// TIA Portal V16 export
// export: Created 2024-12-03T15:41:42.4438673Z, ExportSetting WithDefaults, DisplayName Totally Integrated Automation Portal, DisplayVersion V16 Update 6, DisplayName TIA Portal Version Control Interface, DisplayVersion V16 Update 2, DisplayName TIA Portal Openness, DisplayVersion V16 Update 6, DisplayName TIA Portal Teamcenter Gateway, DisplayVersion V16, DisplayName SINAMICS Startdrive Advanced, DisplayVersion V16 Update 5, DisplayName SINAMICS Startdrive G130, G150, S120, S150, SINAMICS MV, S210, DisplayVersion V16 Update 5, DisplayName SINAMICS Startdrive G110M, G120, G120C, G120D, G120P, G115D, DisplayVersion V16 Update 5, DisplayName STEP 7 Professional, DisplayVersion V16 Update 6, DisplayName STEP 7 Safety, DisplayVersion V16, DisplayName WinCC Advanced / Unified PC, DisplayVersion V16 Update 6
FUNCTION_BLOCK "EC_Cognex_Dataman_Single_FB"   // FB84, SCL
{ S7_Optimized_Access := 'TRUE' }
VERSION : 0.1
// stored: AutoNumber true, IsIECCheckEnabled false, IsRetainMemResEnabled false, MemoryReserve 100, SetENOAutomatically false, UDAEnableTagReadback false
   VAR_INPUT
      I_HwId : HW_ANY;
      I_Result : "COGNEX_DATAMAN_IN_RESULT_UDT";
      I_ResultStatus : "COGNEX_DATAMAN_IN_RESULT_STATUS_UDT";
      I_Status : "COGNEX_DATAMAN_IN_STATUS_UDT";
   END_VAR
   VAR_OUTPUT
      O_Control : "COGNEX_DATAMAN_OUT_CONTROL_UDT";
      O_Trigger : "COGNEX_DATAMAN_OUT_TRIGGER_UDT";
   END_VAR
   VAR_IN_OUT
      IO_Scanner : "COGNEX_DATAMAN_LOGIC_UDT";
   END_VAR
   VAR
      PrevScanId : Int;
      ScanCommand : "SmartBool";
      triggerAuto { S7_SetPoint := 'True'} : "SmartBool";
      triggerManual { S7_SetPoint := 'True'} : "SmartBool";
      NewResultFlag { S7_SetPoint := 'True'} : "SmartBool";
      MissedTrigger { S7_SetPoint := 'True'} : "SmartBool";
      NotConnected { S7_SetPoint := 'True'} : TON_TIME;
      TimeOutDetector { S7_SetPoint := 'True'} : TON_TIME;
      TimeOutTime { S7_SetPoint := 'True'} : Time;
      StartTimeOut { S7_SetPoint := 'True'} : Bool;
      LockReceiveResult : Bool;
      cycleRun { S7_SetPoint := 'True'} : "CycleRun";
      alarmInfo : "AlarmInfo_UDT";
      TimeOutAlarm { S7_SetPoint := 'True'} : Program_Alarm;
      TriggerGuardAlarm { S7_SetPoint := 'True'} : Program_Alarm;
      ScannerNotConnected { S7_SetPoint := 'True'} : Program_Alarm;
      ErrorFromScanner { S7_SetPoint := 'True'} : Program_Alarm;
      SerialBufferOverlfow { S7_SetPoint := 'True'} : Program_Alarm;
   END_VAR
   VAR_TEMP
      T_AppState : "ApplicationState_UDT";
      T_Zone : "ZoneInfo";
      T_NewResult : Bool;
      T_Error : Int;
      dummy : Array[0..5] of Byte;
   END_VAR
BEGIN
   REGION APPSTATE
       #T_Zone := "ApplicationState_DB".ZoneNames[#IO_Scanner.Zone];
       #T_AppState := "ApplicationState_DB".Appstate[#T_Zone.AppStateIndex];
       #cycleRun();
   END_REGION

   REGION STATUS READERS
       #MissedTrigger(I_Sensor := #I_Status.MissedAck);
       #NewResultFlag(I_Sensor := #I_ResultStatus.ResultsAvaileble);
   END_REGION

   REGION Commands

       #triggerAuto(I_Sensor := #IO_Scanner.Cmd.ScanAuto AND #T_AppState.States.AutoModeActivated.State);
       #triggerManual(I_Sensor := #IO_Scanner.Cmd.ScanManual AND #T_AppState.States.ManualModeActivated.State);

       #ScanCommand(I_Sensor := #triggerAuto.O_data.State OR #triggerManual.O_data.State AND NOT #StartTimeOut);

       IF #ScanCommand.O_data.LE AND NOT #StartTimeOut THEN
           #PrevScanId.%B0 := #I_Status.TriggerId_MSB;
           #PrevScanId.%B1 := #I_Status.TriggerId_LSB;
           #PrevScanId := #PrevScanId;
       END_IF;

   END_REGION

   REGION ALARMS

       REGION INIT
           IF NOT #alarmInfo.init OR #IO_Scanner.Name = '' OR #alarmInfo.info = '' OR "HMI_DB".ReloadSettings.signal THEN
               #alarmInfo.init := true;
               #IO_Scanner.Name := "buildObjectName"(I_Symbolname := GetSymbolName(variable := #IO_Scanner, size := 40));
               #alarmInfo.info := "buildAlarmInfo"(I_ZoneIndex := #IO_Scanner.Zone, I_ZoneName := #T_Zone.ZoneName, I_ObjectName := #IO_Scanner.Name);
           END_IF;
       END_REGION

       REGION timeout scanning
           IF #IO_Scanner.ReadingResult.TimeOut_Pulse THEN
               #IO_Scanner.Alarms.TimeOutReading.Active := TRUE;
           END_IF;
           #IO_Scanner.Alarms.TimeOutReading.Active := FALSE;
           #IO_Scanner.Alarms.status.%X0 := #IO_Scanner.Alarms.TimeOutReading.Active;
       END_REGION

       REGION trigger guard
           IF (#triggerAuto.O_data.State
               OR #triggerManual.O_data.State)
               AND #StartTimeOut THEN
               #IO_Scanner.Alarms.TriggerGuard.Active := TRUE;
           END_IF;
           #IO_Scanner.Alarms.status.%X1 := #IO_Scanner.Alarms.TriggerGuard.Active;
       END_REGION

       REGION scanner not connected

           #T_Error := DPRD_DAT(LADDR := #I_HwId, RECORD => #dummy);

           IF #T_Error > 0 THEN
               #IO_Scanner.Alarms.NotConnected.Active := TRUE;
           END_IF;

           #IO_Scanner.Alarms.status.%X2 := #IO_Scanner.Alarms.NotConnected.Active;
       END_REGION

       REGION error from scanner
           IF #I_ResultStatus.GeneralError THEN
               #IO_Scanner.Alarms.ErrorFromScanner.Active := TRUE;
           END_IF;
           #IO_Scanner.Alarms.ErrorFromScanner.Active := FALSE;
           #IO_Scanner.Alarms.status.%X3 := #IO_Scanner.Alarms.ErrorFromScanner.Active;
       END_REGION

       REGION SERIAL BUFFER OVERFLOW
           IF #I_ResultStatus.ResultBufferOverrun THEN
               #IO_Scanner.Alarms.SerialBufferOverFlow.Active := TRUE;
           END_IF;
           #IO_Scanner.Alarms.status.%X4 := #IO_Scanner.Alarms.SerialBufferOverFlow.Active;
       END_REGION

       REGION PROGRAM ALARMS
           IF #cycleRun.O_Cycle = 5 THEN
               #TimeOutAlarm(SIG := #IO_Scanner.Alarms.TimeOutReading.Active,
                             SD_1 := #T_Zone.ZoneName,
                             SD_2 := #IO_Scanner.Name,
                             SD_3 := #alarmInfo.info);
           END_IF;

           IF #cycleRun.O_Cycle = 6 THEN
               #TriggerGuardAlarm(SIG := #IO_Scanner.Alarms.TriggerGuard.Active,
                                  SD_1 := #T_Zone.ZoneName,
                                  SD_2 := #IO_Scanner.Name,
                                  SD_3 := #alarmInfo.info);
           END_IF;

           IF #cycleRun.O_Cycle = 7 THEN
               #ScannerNotConnected(SIG := #IO_Scanner.Alarms.NotConnected.Active,
                                    SD_1 := #T_Zone.ZoneName,
                                    SD_2 := #IO_Scanner.Name,
                                    SD_3 := #alarmInfo.info);
           END_IF;

           IF #cycleRun.O_Cycle = 8 THEN
               #ErrorFromScanner(SIG := #IO_Scanner.Alarms.ErrorFromScanner.Active,
                                 SD_1 := #T_Zone.ZoneName,
                                 SD_2 := #IO_Scanner.Name,
                                 SD_3 := #alarmInfo.info);
           END_IF;

           IF #cycleRun.O_Cycle = 9 THEN
               #SerialBufferOverlfow(SIG := #IO_Scanner.Alarms.SerialBufferOverFlow.Active,
                                     SD_1 := #T_Zone.ZoneName,
                                     SD_2 := #IO_Scanner.Name,
                                     SD_3 := #alarmInfo.info);
           END_IF;

       END_REGION

       IF #IO_Scanner.Alarms.status > 0 THEN
           "ApplicationState_DB".Appstate[#T_Zone.AppStateIndex].Alarms.AlarmActiveInternalPLC := TRUE;
       END_IF;

       IF #T_AppState.Hmi_Buttons.reset.state.State
           OR #IO_Scanner.Cmd.Reset THEN
           #IO_Scanner.Alarms.TimeOutReading.Active := 0;
           #IO_Scanner.Alarms.TriggerGuard.Active := 0;
           #IO_Scanner.Alarms.NotConnected.Active := 0;
           #IO_Scanner.Alarms.ErrorFromScanner.Active := 0;
           #IO_Scanner.Alarms.SerialBufferOverFlow.Active := 0;
       END_IF;

   END_REGION

   REGION Create status

       #IO_Scanner.Status.ManualModeActive := #T_AppState.States.ManualModeActivated.State;
       #IO_Scanner.Status.ReqBusy := #I_ResultStatus.Decoding OR #StartTimeOut;
       #IO_Scanner.Status.ReqDone := NOT #IO_Scanner.Status.ReqBusy;
       #IO_Scanner.Status.ReadyForNewScan := #I_Status.TriggerReady
       AND NOT #ScanCommand.O_data.State;

   END_REGION

   REGION Parse code

       //Reset pulses
       #IO_Scanner.ReadingResult.Barcode_Pulse := '';
       #IO_Scanner.ReadingResult.GoodRead_Pulse := FALSE;
       #IO_Scanner.ReadingResult.BadRead_Pulse := FALSE;
       #IO_Scanner.ReadingResult.TimeOut_Pulse := FALSE;
       #IO_Scanner.ReadingResult.MissedTrigger_Pulse := FALSE;
       #IO_Scanner.ReadingResult.OutOfSync_Pulse := FALSE;
       #IO_Scanner.ReadingResult.NewResult_Pulse := FALSE;

       REGION GOOD READ / BAD READ
           IF #NewResultFlag.O_data.LE
               AND #I_Result.TriggerId = #PrevScanId
               AND NOT #LockReceiveResult THEN

               REGION reset timed out
                   #StartTimeOut := FALSE;
                   #IO_Scanner.ReadingResult.TimeOut := FALSE;
               END_REGION

               REGION Barcode parsing
                   //IF NOT "Simulation_DB".Simulation_On THEN
                   #IO_Scanner.ReadingResult.chars := #I_Result.Barcode;
                   Chars_TO_Strg(Chars := #IO_Scanner.ReadingResult.chars,
                                 pChars := 0,
                                 Cnt := INT_TO_UINT(#I_Result.ResultLength) - 1, //The last char is new line return we don't need this :)
                                 Strg => #IO_Scanner.ReadingResult.Barcode_Pulse);
                   // ELSE
                   //     #IO_Scanner.ReadingResult.Barcode_Pulse := #IO_Scanner.ReadingResult.Barcode;
                   // END_IF;

                   #IO_Scanner.ReadingResult.Barcode := '';
                   #IO_Scanner.ReadingResult.Barcode := #IO_Scanner.ReadingResult.Barcode_Pulse;
               END_REGION

               REGION SIM
                   IF "Simulation_DB".barcode_sim THEN
                       #IO_Scanner.ReadingResult.Barcode_Pulse := 'BarcodeSim';
                       #IO_Scanner.ReadingResult.Barcode := #IO_Scanner.ReadingResult.Barcode_Pulse;
                   END_IF;

               END_REGION

               REGION Good Read / bad read
                   IF #IO_Scanner.ReadingResult.Barcode_Pulse = 'NoRead' THEN
                       #IO_Scanner.ReadingResult.BadRead_Pulse := TRUE;
                   ELSE
                       #IO_Scanner.ReadingResult.GoodRead_Pulse := TRUE;
                   END_IF;
                   #IO_Scanner.ReadingResult.GoodRead := #IO_Scanner.ReadingResult.GoodRead_Pulse;
                   #IO_Scanner.ReadingResult.BadRead := #IO_Scanner.ReadingResult.BadRead_Pulse;
                   #IO_Scanner.ReadingResult.MissedTrigger := FALSE;
                   #IO_Scanner.ReadingResult.OutOfSync := FALSE;
               END_REGION

           END_IF;
       END_REGION

       REGION MISSED TRIGGER
           IF #MissedTrigger.O_data.LE AND NOT #LockReceiveResult THEN
               #IO_Scanner.ReadingResult.GoodRead := FALSE;
               #IO_Scanner.ReadingResult.BadRead := TRUE;
               #IO_Scanner.ReadingResult.MissedTrigger := TRUE;
               #IO_Scanner.ReadingResult.OutOfSync := FALSE;
               #IO_Scanner.ReadingResult.TimeOut := FALSE;

               #IO_Scanner.ReadingResult.MissedTrigger_Pulse := TRUE;

               #IO_Scanner.ReadingResult.Barcode_Pulse := 'MISSED TRIGGER';
               #IO_Scanner.ReadingResult.Barcode := #IO_Scanner.ReadingResult.Barcode_Pulse;
           END_IF;
       END_REGION

       REGION OUT OF SYNC
           IF #NewResultFlag.O_data.LE
               AND #PrevScanId <> #I_Result.TriggerId
               AND NOT #LockReceiveResult
           THEN
               #IO_Scanner.ReadingResult.GoodRead := FALSE;
               #IO_Scanner.ReadingResult.BadRead := TRUE;
               #IO_Scanner.ReadingResult.MissedTrigger := FALSE;
               #IO_Scanner.ReadingResult.OutOfSync := TRUE;
               #IO_Scanner.ReadingResult.TimeOut := FALSE;

               #IO_Scanner.ReadingResult.OutOfSync_Pulse := TRUE;

               #IO_Scanner.ReadingResult.Barcode_Pulse := 'OUT OF SYNC';
               #IO_Scanner.ReadingResult.Barcode := #IO_Scanner.ReadingResult.Barcode_Pulse;
           END_IF;
       END_REGION

       REGION Time out reading result detection

           // Reset-disable time out when scan command is active
           IF #ScanCommand.O_data.LE THEN
               //#StartTimeOut := FALSE;
               #LockReceiveResult := FALSE;
           END_IF;

           // Start time out when FE scan command
           IF #ScanCommand.O_data.FE AND NOT #StartTimeOut AND NOT #I_ResultStatus.ResultsAvaileble THEN
               #StartTimeOut := TRUE;
           END_IF;

           // Reset timer when there is no time out running
           IF NOT #StartTimeOut THEN
               RESET_TIMER(#TimeOutDetector);
           END_IF;

           // Copy time out time for diagnostics
           IF #StartTimeOut THEN
               #IO_Scanner.DiagNostic.ParsingTime := #TimeOutDetector.ET;
           END_IF;

           #TimeOutDetector(IN := #StartTimeOut,
                            PT := #IO_Scanner.Settings.TimeOut);

           // Time out occured :(
           IF #TimeOutDetector.Q THEN
               #StartTimeOut := FALSE;
               RESET_TIMER(#TimeOutDetector);
               #LockReceiveResult := TRUE;
               #IO_Scanner.ReadingResult.GoodRead := FALSE;
               #IO_Scanner.ReadingResult.BadRead := TRUE;
               #IO_Scanner.ReadingResult.BadRead_Pulse := TRUE;
               #IO_Scanner.ReadingResult.TimeOut_Pulse := TRUE;
               #IO_Scanner.ReadingResult.TimeOut := TRUE;
               #IO_Scanner.ReadingResult.Barcode_Pulse := 'Timeout';
               #IO_Scanner.ReadingResult.Barcode := #IO_Scanner.ReadingResult.Barcode_Pulse;
           END_IF;

       END_REGION

       REGION NEW RESULT PULSE
           IF #IO_Scanner.ReadingResult.BadRead_Pulse
               OR #IO_Scanner.ReadingResult.GoodRead_Pulse
               OR #IO_Scanner.ReadingResult.TimeOut_Pulse THEN
               #IO_Scanner.ReadingResult.NewResult_Pulse := True;
           END_IF;
       END_REGION

   END_REGION

   REGION Handle diagnostics

       IF #ScanCommand.O_data.LE THEN
           #IO_Scanner.DiagNostic.Scans += 1;
       END_IF;

       IF #IO_Scanner.ReadingResult.BadRead_Pulse THEN
           #IO_Scanner.DiagNostic.BadReads += 1;
       END_IF;

       IF #IO_Scanner.ReadingResult.GoodRead_Pulse THEN
           #IO_Scanner.DiagNostic.GoodReads += 1;
       END_IF;

       IF #IO_Scanner.ReadingResult.TimeOut_Pulse THEN
           #IO_Scanner.DiagNostic.TimeOuts += 1;
       END_IF;

       IF #IO_Scanner.ReadingResult.MissedTrigger_Pulse THEN
           #IO_Scanner.DiagNostic.MissedTrigger += 1;
       END_IF;

       IF #IO_Scanner.ReadingResult.OutOfSync_Pulse THEN
           #IO_Scanner.DiagNostic.OutOfSync += 1;
       END_IF;

   END_REGION

   REGION OUTPUT CONTROL

       REGION ACK NEW DATA
           #O_Control.ResultsAck := #I_ResultStatus.ResultsAvaileble
           AND NOT #O_Trigger.Trigger;
       END_REGION

       REGION setttings
           #O_Trigger.TriggerEnable := #IO_Scanner.Alarms.status = 0;
       END_REGION

       REGION SENT TRIGGER COMMAND
           #O_Trigger.Trigger := #ScanCommand.O_data.State;

       END_REGION

   END_REGION

   IF #IO_Scanner.Cmd.Reset THEN
       #IO_Scanner.Cmd.Reset := 0;
   END_IF;
END_FUNCTION_BLOCK
